PROGRAM P_InfluxTEST
VAR
	rand 	: DRAND;							// Instance of DRAND function block
    nrand	: LREAL;			
	fValue1	: LREAL;
	fValue2	: LREAL;
	fValue3	: LREAL;
END_VAR

rand();
nrand := rand.Num;
fValue1 := 240.328 + 10 * nrand;
fValue2 := 7.3292 + nrand;
fValue3 := 1113.1975 + 50 * nrand;

END_PROGRAM

(* stored: Version 1.1.0.1, ProductVersion 3.1.4024.11
   POU P_InfluxTEST: Id {d7aa5ba8-4ace-4a8d-81d6-4cbcf65000f1}, SpecialFunc None *)
